{attribute addProperty BoxType "ER3184-0002-0019"}
{attribute addProperty Id "AI_Standard_ChannelAT %I*ARRAY[0..6] OF AI_Standard_Channel_904746A2128160WcStateAT %I*WcState_98A4DF7520.250InfoDataAT %I*InfoData_BC63D37F80100"}
{attribute addProperty CRC "1539253693"}
{attribute addProperty SizeInBites "210"}
{attribute addProperty SizeInBytes "26.25"}
TYPE ER3184_6082EBFD :
STRUCT
	{attribute addProperty Name "AI_Standard_Channel"}
	AI_Standard_Channel : ARRAY[0..6] OF AI_Standard_Channel_904746A2;
	{attribute addProperty Name "WcState"}
	WcState : WcState_98A4DF75;
	{attribute addProperty Name "InfoData"}
	InfoData : InfoData_BC63D37F;
END_STRUCT
END_TYPE

(* stored: Version 1.2.0.0, ProductVersion 3.1.4024.9
   DUT ER3184_6082EBFD: Id {0be318cc-199b-437b-8a55-4e197d500402} *)
